{attribute 'linkalways'} 
FUNCTION GetByteOffset : PVOID
VAR_INPUT
	Structure : ANY;
	Member : ANY_BIT; 
END_VAR

GetByteOffset := Member.pValue - Structure.pValue;

END_FUNCTION

(* stored: Version 1.1.0.1, ProductVersion 3.1.4024.12
   POU GetByteOffset: Id {0efc41c6-3334-4710-9ede-e85597a19f9b}, SpecialFunc None *)
